SUBAPPLICATION OPC_SUB_FIO (* Subapplication Type *)
  (* Standard: 61499-2 *)
  (* Version 1.0, 2022-03-11, Maximilian Scharf *)
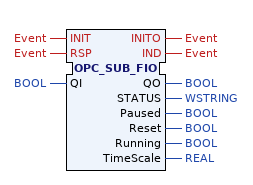
  EVENT_INPUT
    INIT;
    RSP;
  END_EVENT
  EVENT_OUTPUT
    INITO;
    IND;
  END_EVENT
  VAR_INPUT
    QI : BOOL;
  END_VAR
  VAR_OUTPUT
    QO : BOOL;
    STATUS : WSTRING;
    Paused : BOOL;
    Reset : BOOL;
    Running : BOOL;
    TimeScale : REAL;
  END_VAR
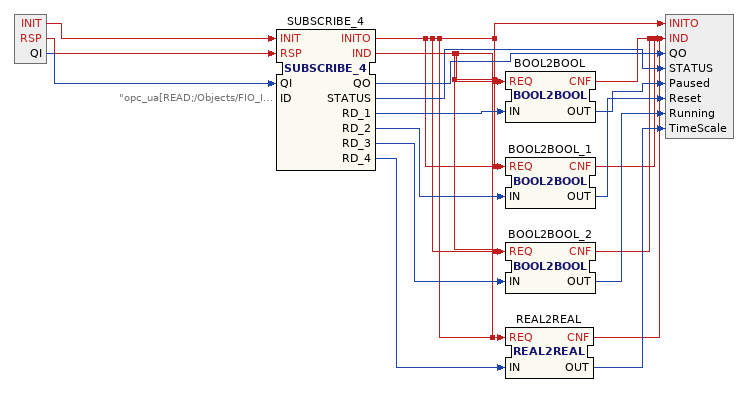
  FBS
    SUBSCRIBE_4 : SUBSCRIBE_4(ID := "opc_ua[READ;/Objects/FIO_I_Paused, 1:s=FIO_I_Paused;/Objects/FIO_I_Reset, 1:s=FIO_I_Reset;/Objects/FIO_I_Running, 1:s=FIO_I_Running;/Objects/FIO_I_TimeScale, 1:s=FIO_I_TimeScale]");
    BOOL2BOOL : BOOL2BOOL;
    BOOL2BOOL_1 : BOOL2BOOL;
    BOOL2BOOL_2 : BOOL2BOOL;
    REAL2REAL : REAL2REAL;
  END_FBS
  EVENT_CONNECTIONS
    INIT TO SUBSCRIBE_4.INIT;
    RSP TO SUBSCRIBE_4.RSP;
    SUBSCRIBE_4.INITO TO INITO;
    SUBSCRIBE_4.IND TO BOOL2BOOL.REQ;
    SUBSCRIBE_4.INITO TO BOOL2BOOL.REQ;
    SUBSCRIBE_4.INITO TO BOOL2BOOL_1.REQ;
    SUBSCRIBE_4.INITO TO BOOL2BOOL_2.REQ;
    SUBSCRIBE_4.INITO TO REAL2REAL.REQ;
    SUBSCRIBE_4.IND TO BOOL2BOOL_1.REQ;
    SUBSCRIBE_4.IND TO BOOL2BOOL_2.REQ;
    SUBSCRIBE_4.IND TO REAL2REAL.REQ;
    BOOL2BOOL.CNF TO IND;
    BOOL2BOOL_1.CNF TO IND;
    BOOL2BOOL_2.CNF TO IND;
    REAL2REAL.CNF TO IND;
  END_CONNECTIONS
  DATA_CONNECTIONS
    QI TO SUBSCRIBE_4.QI;
    SUBSCRIBE_4.QO TO QO;
    SUBSCRIBE_4.STATUS TO STATUS;
    SUBSCRIBE_4.RD_1 TO BOOL2BOOL.IN;
    BOOL2BOOL.OUT TO Paused;
    SUBSCRIBE_4.RD_2 TO BOOL2BOOL_1.IN;
    BOOL2BOOL_1.OUT TO Reset;
    SUBSCRIBE_4.RD_3 TO BOOL2BOOL_2.IN;
    BOOL2BOOL_2.OUT TO Running;
    REAL2REAL.OUT TO TimeScale;
    SUBSCRIBE_4.RD_4 TO REAL2REAL.IN;
  END_CONNECTIONS
END_SUBAPPLICATION
